PROGRAM MAIN
VAR
END_VAR

(*
fb_TV2K0_VFS_1(
	i_xPMPS_OK:= TRUE, 
	i_xExt_OK:= TRUE, 
	iq_stValve=>,
	io_fbFFHWO:= g_FastFaultOutput2
);
*)

END_PROGRAM

(* stored: Version 1.1.0.1, ProductVersion 3.1.4024.2
   POU MAIN: Id {400798bf-4b47-4e69-b0b8-9446fd0f52d0}, SpecialFunc None *)
